// TIA Portal V20 export
DATA_BLOCK "DB_NordSetPoint"   // DB48
// stored: Access Published, MemoryReserve 100, Namespace LineD1
   VAR
      Line : Struct
         D1 : Struct   // -(0 - 16000) -> (CW: 0 - 100%) || +(0 - 16000) (CCW: 0 - 100%) || freq. has been set via NORDCON
            Conveyor : Array[_.minD1.._.maxD1] of DInt;
         END_STRUCT;
      END_STRUCT;
   END_VAR
BEGIN
END_DATA_BLOCK
